# EPICS substitutions: BL99I-LCH-IOC-01App/Db/motorTest.substitutions
file $(PMAC)/db/pmacController.template
{
pattern { PORT, P, NAXES, TIMEOUT, FEEDRATE, CSG0, CSG1, CSG2, CSG3, CSG4, CSG5, CSG6, CSG7 }
    { "BRICK1", "BL99I-LCH-STEP-01", "8", "4", "100", "", "", "", "", "", "", "", "" }
}

file $(PMAC)/db/pmacStatus.template
{
pattern { PORT, P }
    { "BRICK1", "BL99I-LCH-STEP-01" }
}

file $(PMAC)/db/pmacCSS.template
{
pattern { NAME, P, Description, ControlIP, ControlPort, ControlMode }
    { "BRICK1", "BL99I-LCH-STEP-01", "None", "None", "None", "None" }
}

file $(PMAC)/db/pmacStatusAxis.template
{
pattern { PMAC, AXIS, PORT }
    { "BL99I-LCH-STEP-01", "1", "BRICK1" }
    { "BL99I-LCH-STEP-01", "2", "BRICK1" }
    { "BL99I-LCH-STEP-01", "3", "BRICK1" }
    { "BL99I-LCH-STEP-01", "4", "BRICK1" }
    { "BL99I-LCH-STEP-01", "5", "BRICK1" }
    { "BL99I-LCH-STEP-01", "6", "BRICK1" }
    { "BL99I-LCH-STEP-01", "7", "BRICK1" }
    { "BL99I-LCH-STEP-01", "8", "BRICK1" }
}

file $(PMAC)/db/dls_pmac_asyn_motor.template
{
pattern { P,                        M,          PORT,       ADDR,   DESC,   MRES,       VELO,   PREC, EGU, TWV, DTYP,           DIR,    VBAS, VMAX, ACCL, BDST, BVEL,   BACC,   DHLM, DLLM, HLM, LLM, HLSV, INIT, SREV, RRES, ERES, JAR, UEIP, URIP, RDBL, RLNK, RTRY, DLY, OFF, RDBD, FOFF, ADEL, NTM, FEHIGH, FEHIHI, FEHHSV, FEHSV, SCALE, HOMEVIS, HOMEVISSTR, name, alh, gda_name, gda_desc, SPORT, HOME, PMAC, ALLOW_HOMED_SET }
        { "BL99I-LCH-STEP-01:A1",   ":XPLUS",   "BRICK1",   "1",    "X+",   "0.000001", "0.5",  "5", "mm", "1", "asynMotor",    "0",    "0", "0.5", "0.5", "0", "0",    "",     "10", "-10", "10", "-10", "MAJOR", "", "1000", "", "", "", "0", "0", "", "", "0", "0", "", "", "0", "0", "1", "0", "0", "NO_ALARM", "NO_ALARM", "1", "1", "Use motor summary screen", "A1", "None", "", "$(DESC)", "BRICK1port", "$(P)", "BL99I-LCH-STEP-01", "#" }
}
